// TIA Portal V15.1 export
// export: Created 2024-05-17T05:38:17.1370677Z, ExportSetting WithDefaults, DisplayName Totally Integrated Automation Portal, DisplayVersion V15.1 Update 5, DisplayName TIA Portal Openness, DisplayVersion V15.1 Update 5, DisplayName SINAMICS Startdrive Advanced, DisplayVersion V15.1, DisplayName G130, G150, S120, S150, SINAMICS MV, S210, DisplayVersion V15.1, DisplayName G110M, G120, G120C, G120D, G120P, DisplayVersion V15.1, DisplayName STEP 7 Professional, DisplayVersion V15.1 Update 5, DisplayName STEP 7 Safety, DisplayVersion V15.1, DisplayName WinCC Professional, DisplayVersion V15.1 Update 5, DisplayName SIMATIC Visualization Architect, DisplayVersion V15.1
DATA_BLOCK "_209220ZS01PNIODiag"   // DB374
{ S7_Optimized_Access := 'FALSE' }
AUTHOR : VCC
VERSION : 0.1
// stored: AutoNumber false, DBAccessibleFromOPCUA true, IsOnlyStoredInLoadMemory false, IsWriteProtectedInAS false
   VAR RETAIN
      "AA_209220AS10-JW50" { ExternalAccessible := 'False'; ExternalVisible := 'False'; ExternalWritable := 'False'} : Bool;   // Profinet device don't exist - ET200sp I/O - Busnode 220AS10 - node 50
      "AA_209220AX01-JW51" { ExternalAccessible := 'False'; ExternalVisible := 'False'; ExternalWritable := 'False'} : Bool;   // Profinet device don't exist - ET200sp I/O - Busnode 220AX01 - node 51
      "AA_209220AS11-JW52" { ExternalAccessible := 'False'; ExternalVisible := 'False'; ExternalWritable := 'False'} : Bool;   // Profinet device don't exist - ET200sp I/O - Busnode 220AS11 - node 52
      "AA_209220AX02-JW53" { ExternalAccessible := 'False'; ExternalVisible := 'False'; ExternalWritable := 'False'} : Bool;   // Profinet device don't exist - ET200sp I/O - Busnode 220AX02 - node 53
      "AC_209220CWP10-JX54" { ExternalAccessible := 'False'; ExternalVisible := 'False'; ExternalWritable := 'False'} : Bool;   // Profinet device don't exist - ET200eco I/O - Module 220CWP10 - node 54
      "AC_209220CWP10-JX55" { ExternalAccessible := 'False'; ExternalVisible := 'False'; ExternalWritable := 'False'} : Bool;   // Profinet device don't exist - ET200eco I/O - Module 220CWP10 - node 55
      "AC_209220CWP20-JX56" { ExternalAccessible := 'False'; ExternalVisible := 'False'; ExternalWritable := 'False'} : Bool;   // Profinet device don't exist - ET200eco I/O - Module 220CWP20 - node 56
      "AC_209220CWP20-JX57" { ExternalAccessible := 'False'; ExternalVisible := 'False'; ExternalWritable := 'False'} : Bool;   // Profinet device don't exist - ET200eco I/O - Module 220CWP20 - node 57
      "AA_209220AS20-JW58" { ExternalAccessible := 'False'; ExternalVisible := 'False'; ExternalWritable := 'False'} : Bool;   // Profinet device don't exist - ET200sp I/O - Busnode 220AS20 - node 58
      "AB_209000AK04M1-UE140" { ExternalAccessible := 'False'; ExternalVisible := 'False'; ExternalWritable := 'False'} : Bool;   // Profinet device don't exist - MoviDrive - 220CR21M1 - node 140
      "AB_209000AK04M4-UE141" { ExternalAccessible := 'False'; ExternalVisible := 'False'; ExternalWritable := 'False'} : Bool;   // Profinet device don't exist - MoviDrive - 220CS22M4(Power) - node 141
      "AB_209000AK04M4-UE142" { ExternalAccessible := 'False'; ExternalVisible := 'False'; ExternalWritable := 'False'} : Bool;   // Profinet device don't exist - MoviDrive - 220CS22M4(Brake) - node 142
      "AB_209000AK04M1-UE143" { ExternalAccessible := 'False'; ExternalVisible := 'False'; ExternalWritable := 'False'} : Bool;   // Profinet device don't exist - MoviDrive - 220CR23M1 - node 143
      "AB_209220CHB21M14-UE144" { ExternalAccessible := 'False'; ExternalVisible := 'False'; ExternalWritable := 'False'} : Bool;   // Profinet device don't exist - MoviFit - 220CHB21M14 - node 144
      "AA_209220Field-JW222" { ExternalAccessible := 'False'; ExternalVisible := 'False'; ExternalWritable := 'False'} : Bool;   // Profinet device don't exist - Field Switch - Safety Zone 220 - node 222
      "AA_209220Field-JW232" { ExternalAccessible := 'False'; ExternalVisible := 'False'; ExternalWritable := 'False'} : Bool;   // Profinet device don't exist - Field Switch - Safety Zone 220 - node 232
      "AC_209220AS10-JW50Fault" { ExternalAccessible := 'False'; ExternalVisible := 'False'; ExternalWritable := 'False'} : Bool;   // Faulty profinet device -> For more detail information look for N.A. alarms in the alarmlist - ET200sp I/O - Busnode 220AS10 - node 50
      "AC_209220AX01-JW51Fault" { ExternalAccessible := 'False'; ExternalVisible := 'False'; ExternalWritable := 'False'} : Bool;   // Faulty profinet device -> For more detail information look for N.A. alarms in the alarmlist - ET200sp I/O - Busnode 220AX01 - node 51
      "AC_209220AS11-JW52Fault" { ExternalAccessible := 'False'; ExternalVisible := 'False'; ExternalWritable := 'False'} : Bool;   // Faulty profinet device -> For more detail information look for N.A. alarms in the alarmlist - ET200sp I/O - Busnode 220AS11 - node 52
      "AC_209220AX02-JW53Fault" { ExternalAccessible := 'False'; ExternalVisible := 'False'; ExternalWritable := 'False'} : Bool;   // Faulty profinet device -> For more detail information look for N.A. alarms in the alarmlist - ET200sp I/O - Busnode 220AX02 - node 53
      "AC_209220CWP10-JX54Fault" { ExternalAccessible := 'False'; ExternalVisible := 'False'; ExternalWritable := 'False'} : Bool;   // Faulty profinet device -> For more detail information look for N.A. alarms in the alarmlist - ET200eco I/O - Module 220CWP10 - node 54
      "AC_209220CWP10-JX55Fault" { ExternalAccessible := 'False'; ExternalVisible := 'False'; ExternalWritable := 'False'} : Bool;   // Faulty profinet device -> For more detail information look for N.A. alarms in the alarmlist - ET200eco I/O - Module 220CWP10 - node 55
      "AC_209220CWP20-JX56Fault" { ExternalAccessible := 'False'; ExternalVisible := 'False'; ExternalWritable := 'False'} : Bool;   // Faulty profinet device -> For more detail information look for N.A. alarms in the alarmlist - ET200eco I/O - Module 220CWP20 - node 56
      "AC_209220CWP20-JX57Fault" { ExternalAccessible := 'False'; ExternalVisible := 'False'; ExternalWritable := 'False'} : Bool;   // Faulty profinet device -> For more detail information look for N.A. alarms in the alarmlist - ET200eco I/O - Module 220CWP20 - node 57
      "AC_209220AS20-JW58Fault" { ExternalAccessible := 'False'; ExternalVisible := 'False'; ExternalWritable := 'False'} : Bool;   // Faulty profinet device -> For more detail information look for N.A. alarms in the alarmlist - ET200sp I/O - Busnode 220AS20 - node 58
      "AC_209000AK04M1-UE140Fault" { ExternalAccessible := 'False'; ExternalVisible := 'False'; ExternalWritable := 'False'} : Bool;   // Faulty profinet device -> For more detail information look for N.A. alarms in the alarmlist - MoviDrive - 220CR21M1 - node 140
      "AC_209000AK04M4-UE141Fault" { ExternalAccessible := 'False'; ExternalVisible := 'False'; ExternalWritable := 'False'} : Bool;   // Faulty profinet device -> For more detail information look for N.A. alarms in the alarmlist - MoviDrive - 220CS22M4(Power) - node 141
      "AC_209000AK04M4-UE142Fault" { ExternalAccessible := 'False'; ExternalVisible := 'False'; ExternalWritable := 'False'} : Bool;   // Faulty profinet device -> For more detail information look for N.A. alarms in the alarmlist - MoviDrive - 220CS22M4(Brake) - node 142
      "AC_209000AK04M1-UE143Fault" { ExternalAccessible := 'False'; ExternalVisible := 'False'; ExternalWritable := 'False'} : Bool;   // Faulty profinet device -> For more detail information look for N.A. alarms in the alarmlist - MoviDrive - 220CR23M1 - node 143
      "AC_209220CHB21M14-UE144Fault" { ExternalAccessible := 'False'; ExternalVisible := 'False'; ExternalWritable := 'False'} : Bool;   // Faulty profinet device -> For more detail information look for N.A. alarms in the alarmlist - MoviFit - 220CHB21M14 - node 144
      "AC_209220Field-JW222Fault" { ExternalAccessible := 'False'; ExternalVisible := 'False'; ExternalWritable := 'False'} : Bool;   // Faulty profinet device -> For more detail information look for N.A. alarms in the alarmlist - Field Switch - Safety Zone 220 - node 222
      "AC_209220Field-JW232Fault" { ExternalAccessible := 'False'; ExternalVisible := 'False'; ExternalWritable := 'False'} : Bool;   // Faulty profinet device -> For more detail information look for N.A. alarms in the alarmlist - Field Switch - Safety Zone 220 - node 232
      "209220AS10-JW50AlarmABCondition" { ExternalAccessible := 'False'; ExternalVisible := 'False'; ExternalWritable := 'False'} : Bool;   // Alarm AB condition
      "209220AX01-JW51AlarmABCondition" { ExternalAccessible := 'False'; ExternalVisible := 'False'; ExternalWritable := 'False'} : Bool;   // Alarm AB condition
      "209220AS11-JW52AlarmABCondition" { ExternalAccessible := 'False'; ExternalVisible := 'False'; ExternalWritable := 'False'} : Bool;   // Alarm AB condition
      "209220AX02-JW53AlarmABCondition" { ExternalAccessible := 'False'; ExternalVisible := 'False'; ExternalWritable := 'False'} : Bool;   // Alarm AB condition
      "209220AS20-JW58AlarmABCondition" { ExternalAccessible := 'False'; ExternalVisible := 'False'; ExternalWritable := 'False'} : Bool;   // Alarm AB condition
      "209000AK04M1-UE140AlarmABCondition" { ExternalAccessible := 'False'; ExternalVisible := 'False'; ExternalWritable := 'False'} : Bool;   // Alarm AB condition
      "209000AK04M4-UE141AlarmABCondition" { ExternalAccessible := 'False'; ExternalVisible := 'False'; ExternalWritable := 'False'} : Bool;   // Alarm AB condition
      "209000AK04M4-UE142AlarmABCondition" { ExternalAccessible := 'False'; ExternalVisible := 'False'; ExternalWritable := 'False'} : Bool;   // Alarm AB condition
      "209000AK04M1-UE143AlarmABCondition" { ExternalAccessible := 'False'; ExternalVisible := 'False'; ExternalWritable := 'False'} : Bool;   // Alarm AB condition
      "209220CHB21M14-UE144AlarmABCondition" { ExternalAccessible := 'False'; ExternalVisible := 'False'; ExternalWritable := 'False'} : Bool;   // Alarm AB condition
      "209220Field-JW222AlarmABCondition" { ExternalAccessible := 'False'; ExternalVisible := 'False'; ExternalWritable := 'False'} : Bool;   // Alarm AB condition
      "209220Field-JW232AlarmABCondition" { ExternalAccessible := 'False'; ExternalVisible := 'False'; ExternalWritable := 'False'} : Bool;   // Alarm AB condition
      "H_209220AS10-JW50IAnim" : Word;   // HMI Animation of the icon
      "H_209220AX01-JW51IAnim" : Word;   // HMI Animation of the icon
      "H_209220AS11-JW52IAnim" : Word;   // HMI Animation of the icon
      "H_209220AX02-JW53IAnim" : Word;   // HMI Animation of the icon
      "H_209220CWP10-JX54IAnim" : Word;   // HMI Animation of the icon
      "H_209220CWP10-JX55IAnim" : Word;   // HMI Animation of the icon
      "H_209220CWP20-JX56IAnim" : Word;   // HMI Animation of the icon
      "H_209220CWP20-JX57IAnim" : Word;   // HMI Animation of the icon
      "H_209220AS20-JW58IAnim" : Word;   // HMI Animation of the icon
      "H_209000AK04M1-UE140IAnim" : Word;   // HMI Animation of the icon
      "H_209000AK04M4-UE141IAnim" : Word;   // HMI Animation of the icon
      "H_209000AK04M4-UE142IAnim" : Word;   // HMI Animation of the icon
      "H_209000AK04M1-UE143IAnim" : Word;   // HMI Animation of the icon
      "H_209220CHB21M14-UE144IAnim" : Word;   // HMI Animation of the icon
      "H_209220Field-JW222IAnim" : Word;   // HMI Animation of the icon
      "H_209220Field-JW232IAnim" : Word;   // HMI Animation of the icon
      "H_209220AS10-JW50IAnim2" : Word;   // HMI Animation of the icon
      "H_209220AX01-JW51IAnim2" : Word;   // HMI Animation of the icon
      "H_209220AS11-JW52IAnim2" : Word;   // HMI Animation of the icon
      "H_209220AX02-JW53IAnim2" : Word;   // HMI Animation of the icon
      "H_209220CWP10-JX54IAnim2" : Word;   // HMI Animation of the icon
      "H_209220CWP10-JX55IAnim2" : Word;   // HMI Animation of the icon
      "H_209220CWP20-JX56IAnim2" : Word;   // HMI Animation of the icon
      "H_209220CWP20-JX57IAnim2" : Word;   // HMI Animation of the icon
      "H_209220AS20-JW58IAnim2" : Word;   // HMI Animation of the icon
      "H_209000AK04M1-UE140IAnim2" : Word;   // HMI Animation of the icon
      "H_209000AK04M4-UE141IAnim2" : Word;   // HMI Animation of the icon
      "H_209000AK04M4-UE142IAnim2" : Word;   // HMI Animation of the icon
      "H_209000AK04M1-UE143IAnim2" : Word;   // HMI Animation of the icon
      "H_209220CHB21M14-UE144IAnim2" : Word;   // HMI Animation of the icon
      "H_209220Field-JW222IAnim2" : Word;   // HMI Animation of the icon
      "H_209220Field-JW232IAnim2" : Word;   // HMI Animation of the icon
      H_IAnim : Word;   // Icon Animation / Animation
      H_Anim : Word;   // Animation
      H_DBnr : Int;   // DB number
      AlarmA { ExternalAccessible := 'False'; ExternalVisible := 'False'; ExternalWritable := 'False'} : Bool;   // Summary Alarm A
      AlarmB { ExternalAccessible := 'False'; ExternalVisible := 'False'; ExternalWritable := 'False'} : Bool;   // Summary Alarm B
      AlarmC { ExternalAccessible := 'False'; ExternalVisible := 'False'; ExternalWritable := 'False'} : Bool;   // Summary Alarm C
      AlarmD { ExternalAccessible := 'False'; ExternalVisible := 'False'; ExternalWritable := 'False'} : Bool;   // Summary Alarm D
      AlarmABCondition { ExternalAccessible := 'False'; ExternalVisible := 'False'; ExternalWritable := 'False'} : Bool;   // Alarm AB Condition
   END_VAR
BEGIN
END_DATA_BLOCK
